# B&R Automation Studio project new
Automation Studio 4.5.2.102

## Configuration OG1

### Task classes (Cpu.sw)
```
Cyclic#4:
  Program <- Program.prg
```

## Logical view

### Library Logical/Libraries/Library

#### Library.fun
```iecst
{REDUND_ERROR} {REDUND_UNREPLICABLE} FUNCTION_BLOCK FB_Regulator (*TODO: Add your comment here*) (*$GROUP=User,$CAT=User,$GROUPICON=User.png,$CATICON=User.png*)
	VAR_INPUT
		e : {REDUND_UNREPLICABLE} REAL;
	END_VAR
	VAR_OUTPUT
		u : {REDUND_UNREPLICABLE} REAL;
	END_VAR
	VAR
		integrator : {REDUND_UNREPLICABLE} FB_Integrator;
		k_p : {REDUND_UNREPLICABLE} REAL;
		k_i : {REDUND_UNREPLICABLE} REAL;
		iyOld : {REDUND_UNREPLICABLE} REAL;
		max_abs_value : {REDUND_UNREPLICABLE} REAL;
		dt : {REDUND_UNREPLICABLE} REAL;
	END_VAR
END_FUNCTION_BLOCK

{REDUND_ERROR} {REDUND_UNREPLICABLE} FUNCTION_BLOCK FB_Motor (*TODO: Add your comment here*) (*$GROUP=User,$CAT=User,$GROUPICON=User.png,$CATICON=User.png*)
	VAR_INPUT
		u : {REDUND_UNREPLICABLE} REAL;
	END_VAR
	VAR_OUTPUT
		w : {REDUND_UNREPLICABLE} REAL;
		phi : {REDUND_UNREPLICABLE} REAL;
	END_VAR
	VAR
		integrator : {REDUND_UNREPLICABLE} FB_Integrator;
		Tm : {REDUND_UNREPLICABLE} REAL;
		ke : {REDUND_UNREPLICABLE} REAL;
		dt : {REDUND_UNREPLICABLE} REAL;
	END_VAR
END_FUNCTION_BLOCK

{REDUND_ERROR} {REDUND_UNREPLICABLE} FUNCTION_BLOCK FB_Integrator (*TODO: Add your comment here*) (*$GROUP=User,$CAT=User,$GROUPICON=User.png,$CATICON=User.png*)
	VAR_INPUT
		in : {REDUND_UNREPLICABLE} REAL;
	END_VAR
	VAR_OUTPUT
		out : {REDUND_UNREPLICABLE} REAL;
	END_VAR
	VAR
		dt : {REDUND_UNREPLICABLE} REAL;
	END_VAR
END_FUNCTION_BLOCK
```

#### FB_Integrator.c
```c
#include <bur/plctypes.h>
#ifdef __cplusplus
	extern "C"
	{
#endif
	#include "Library.h"
#ifdef __cplusplus
	};
#endif
/* TODO: Add your comment here */
void FB_Integrator(struct FB_Integrator* inst)
{
	/*TODO: Add your code here*/
	//inst->out=inst->in*inst->dt+inst->out;
	inst->out+=inst->in;

}
```

#### FB_Motor.c
```c
#include <bur/plctypes.h>
#ifdef __cplusplus
	extern "C"
	{
#endif
	#include "Library.h"
#ifdef __cplusplus
	};
#endif
/* TODO: Add your comment here */
void FB_Motor(struct FB_Motor* inst)
{
	inst->integrator.in = (inst->u/inst->ke)*(inst->dt/inst->Tm);
	inst->w=inst->integrator.out-inst->u;
	inst->integrator.in= inst->w*inst->dt;
	inst->phi = inst->integrator.out;

}
```

#### FB_Regulator.c
```c
#include <bur/plctypes.h>
#ifdef __cplusplus
	extern "C"
	{
#endif
	#include "Library.h"
#ifdef __cplusplus
	};
#endif
/* TODO: Add your comment here */
void FB_Regulator(struct FB_Regulator* inst)
{
	float BON(float x)
		{
		if(x>inst->max_abs_value)
		{
			return inst->max_abs_value;
		}
		else
			return x;
			}
	inst->integrator.in=inst->e*inst->k_i*inst->dt+inst->iyOld;
	inst->u=BON((BON(inst->e*inst->k_p)+inst->integrator.out));
	inst->iyOld=-(BON(inst->e*inst->k_p+inst->integrator.out)+BON((BON(inst->e*inst->k_p)+inst->integrator.out));

}
```

### Program Logical/Program

#### Variables.var
```iecst
VAR
	speed : REAL;
	enable : BOOL;
	count : INT;
	fb_motor : {REDUND_UNREPLICABLE} FB_Motor;
	fb_regulator : {REDUND_UNREPLICABLE} FB_Regulator;
	fb_integrator : {REDUND_UNREPLICABLE} FB_Integrator;
	fb_motor2 : {REDUND_UNREPLICABLE} FB_Motor;
END_VAR
```

#### Main.c
```c
#include <bur/plctypes.h>

#ifdef _DEFAULT_INCLUDES
	#include <AsDefault.h>
#endif

void _INIT ProgramInit(void)
{
	fb_motor.dt=0.01;
	fb_motor.ke=2;
	fb_motor.Tm=0.4;
	fb_motor.integrator.dt=0.01;
	fb_motor2.dt=0.01;
	fb_motor2.ke=2;
	fb_motor2.Tm=0.4;
	fb_motor2.integrator.dt=0.01;
	fb_regulator.dt=0.01;
	fb_regulator.k_p=0.0064;
	fb_regulator.k_i=0.16;
	fb_regulator.max_abs_value=24;
	fb_regulator.integrator.dt=0.01;
	enable=1;
	count=0;

}

void _CYCLIC ProgramCyclic(void)
{
	if(enable)
	{
		count+=10;
		if(count<=1000)
		{
			speed=0;
		}
		else
		{ speed=6;
			if(count>=5000)
			{
				count=0;
			}
		}

		}
	fb_regulator.e=speed - fb_motor.w;
	fb_motor2.u=speed;
	//FB_Regulator(&fb_regulator);
	fb_motor.u=fb_regulator.u;
//	FB_Motor(&fb_motor);
  //  FB_Motor(&fb_motor2);

}

void _EXIT ProgramExit(void)
{

}
```
